PROGRAM MAIN
VAR
END_VAR

ModelExecution();

END_PROGRAM

(* stored: Version 1.1.0.1, ProductVersion 3.1.4024.4
   POU MAIN: Id {7b0b13c0-74fe-4c25-a1f3-9f3e4614e0b1}, SpecialFunc None *)
